// Mitsubishi GX Works2 project: test   PLC: FX1N/FX1NC

PROGRAM MAIN
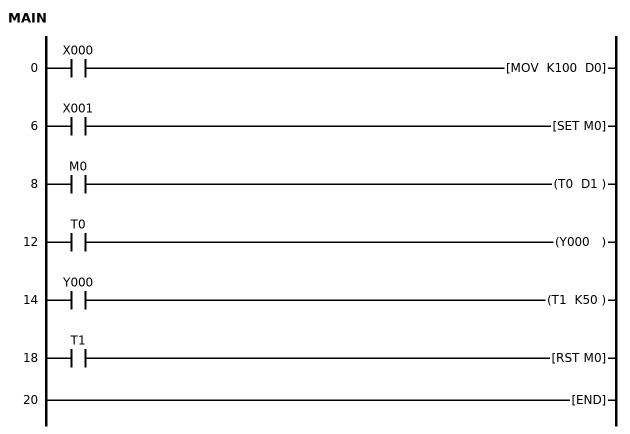
0     LD      X000
      MOV     K100 D0
6     LD      X001
      SET     M0
8     LD      M0
      OUT     T0 D1
12    LD      T0
      OUT     Y000
14    LD      Y000
      OUT     T1 K50
18    LD      T1
      RST     M0
20    END
END_PROGRAM
